{attribute 'pack_mode' := '1'}
    {attribute 'OPC.UA.DA' := '1'}
    {attribute 'OPC.UA.DA.StructuredType' := '1'}
    (*
    ST_RW_KwDeviceInfoGeneric_HMI_IgnitionExp
    ==================================================
    Generated from Ignition UDT: RW_KW_Device_Info_Generic
    Total tags: 8
    Generated on: 2025-09-15 12:56:43
    *)
    TYPE ST_RW_KwDeviceInfoGeneric_HMI_IgnitionExp :
    STRUCT
        {attribute 'OPC.UA.DA' := '1'}
        {attribute 'OPC.UA.DA.Access' := '1'}
        KW_Device_Error : BOOL := FALSE;		// Read-only tag
        {attribute 'OPC.UA.DA' := '1'}
        {attribute 'OPC.UA.DA.Access' := '1'}
        KW_Device_ScanRateMs : DINT := 0;		// Read-only tag
        {attribute 'OPC.UA.DA' := '1'}
        {attribute 'OPC.UA.DA.Access' := '1'}
        KW_Device_Enabled : BOOL := FALSE;		// Read-only tag
        {attribute 'OPC.UA.DA' := '1'}
        {attribute 'OPC.UA.DA.Access' := '1'}
        KW_Device_Description : STRING := '';		// Read-only tag
        {attribute 'OPC.UA.DA' := '1'}
        {attribute 'OPC.UA.DA.Access' := '1'}
        KW_Device_ActiveTagCount : DINT := 0;		// Read-only tag

        {attribute 'OPC.UA.DA' := '1'}
        {attribute 'OPC.UA.DA.Access' := '1'}
        KW_Device_SecondsInError : SINT := 0;		// Read-only tag
        {attribute 'OPC.UA.DA' := '1'}
        {attribute 'OPC.UA.DA.Access' := '1'}
        IPAddress : STRING := '';		// Read-only tag
        {attribute 'OPC.UA.DA' := '1'}
        {attribute 'OPC.UA.DA.Access' := '1'}
        KW_Device_ScanMode : STRING := '';		// Read-only tag
    END_STRUCT
    END_TYPE

(* stored: Version 1.1.0.1
   DUT ST_RW_KwDeviceInfoGeneric_HMI_IgnitionExp: Id {cebfa875-b8e5-49e8-8522-063c732f4e7c} *)
